// This function has been automatically generated from the project information.
{attribute 'signature_flag' := '1073741824'}
{attribute 'TcGenerated'}
{attribute 'no-analysis'}
FUNCTION F_GetTitle : WSTRING
VAR_INPUT
	
END_VAR

F_GetTitle := "protobuf";

END_FUNCTION

(* stored: Version 1.1.0.1
   POU F_GetTitle: Id {949aaccc-af20-4dd4-8fe7-99b4090b12e0}, SpecialFunc None *)
